(* PLC project Tc2_Utilities.UTF8_TO_WSTRING Demo, tc3-libraries-kb TwinCAT 3.1 *)
(* stored: creationDateTime 2026-05-10T16:00:00, modificationDateTime 2026-05-10T16:00:00 *)

PROGRAM P_Demo_UTF8_TO_WSTRING
  VAR
    rResult : BOOL;  (* UTF8_TO_WSTRING 返回值 *)
    bRun : BOOL;  (* 触发一次调用 *)
    sUtf8 : STRING;  (* 测试用本地变量 *)
    wsOut : WSTRING;  (* 测试用本地变量 *)
    nDstLen : UDINT;  (* 测试用本地变量 *)
  END_VAR

            // ============================================================
// Tc2_Utilities.UTF8_TO_WSTRING 演示程序（FUNCTION）
// ============================================================
// 验证步骤：
//   1. 引用 Tc2_Utilities
//   2. 编译 + 登录
//   3. 强制 bRun := TRUE 一个周期
//   4. 在线监视 rResult / 各 demo 变量
// ============================================================

sUtf8 := sLiteral_TO_UTF8('café');
IF bRun THEN
    rResult := UTF8_TO_WSTRING(pDstWSTRING := ADR(wsOut), pSrcUTF8 := ADR(sUtf8), nDstSize := SIZEOF(wsOut), nDstLen => nDstLen);
    bRun := FALSE;
END_IF;

          
END_PROGRAM
